FUNCTION DegToRad : LREAL
VAR_INPUT
    degrees : LREAL;
END_VAR
VAR
END_VAR

DegToRad := degrees / 180.0 * PI;

END_FUNCTION

(* stored: Version 1.1.0.1, ProductVersion 3.1.4018.2
   POU DegToRad: Id {426384a9-b569-4629-8dea-e9ae7f0889eb}, SpecialFunc None *)
